// TIA Portal V20 export
TYPE "LER_typePartDataEm5"
// stored: Access Published
   STRUCT
      cathodeMainPnP1 : "LER_typePartData";
      cathodeAlignTable : "LER_typePartData";
      cathodeMainPnP2 : "LER_typePartData";
      cathodeAlignVision : "LER_typeVisionAlignData";
   END_STRUCT;
END_TYPE
